TYPE TypeTestStruct :
STRUCT
	seed : UDINT;
	bool_var : BOOL;
	sint_var : SINT;
	usint_var : USINT;
	byte_var : BYTE;
	int_var : INT;
	uint_var : UINT;
	word_var : WORD;
	dint_var : DINT;
	udint_var : UDINT;
	dword_var : DWORD;
	lint_var : LINT;
	ulint_var : ULINT;
	lword_var : LWORD;
	real_var : REAL;
	lreal_var : LREAL;
	time_var : TIME;
	tod_var : TOD;
	date_var : DATE;
	dt_var : DT;
	//ltime_var : LTIME;
	//ltod_var : LTOD;
	//ldate_var : LDATE;
	//ldt_var : LDT;
	string_var : STRING(255);
END_STRUCT
END_TYPE

(* stored: Version 1.1.0.1, ProductVersion 3.1.4024.13
   DUT TypeTestStruct: Id {345335e9-ce33-4f05-894a-754f51203bff} *)
